Staubli VAL3: loadmaster2.pgx

program loadmaster2(string x_sMasterFile2 (dimensions=1))
begin
  if master:libLoad(x_sMasterFile2)<0
    popUpMsg("nO ok")
  endIf
  frmaster[2].trsf=master:tTool.trsf
  //取个数
  nsize[2]=size(master:ptRoutingPath)
  //存个数
  resize(pdemo2,1,nsize[2])
  //保存程序
  master:libSave()
end
